// TIA Portal V16 export
// export: Created 2024-05-10T06:46:43.3869042Z, ExportSetting WithDefaults, DisplayName Totally Integrated Automation Portal, DisplayVersion V16, DisplayName TIA Portal Version Control Interface, DisplayVersion V16, DisplayName TIA Portal Openness, DisplayVersion V16, DisplayName STEP 7 Professional, DisplayVersion V16, DisplayName STEP 7 Safety, DisplayVersion V16, DisplayName WinCC Professional, DisplayVersion V16
DATA_BLOCK "K06_动作_DB"   // DB6
VERSION : 0.1
// stored: AutoNumber true, DBAccessibleFromOPCUA true, InstanceOfName K06_动作, InstanceOfType FB
"K06_动作"
   // VAR
   //    INV_Time1 : IEC_TIMER;
   //    INV_Time2 : IEC_TIMER;
   //    F100_Val_Instance1 { S7_SetPoint := 'True'} : "F100_Val";
   //    F100_Val_Instance2 { S7_SetPoint := 'True'} : "F100_Val";
   //    F100_Val_Instance3 { S7_SetPoint := 'True'} : "F100_Val";
   //    F100_Val_Instance4 { S7_SetPoint := 'True'} : "F100_Val";
   //    F100_Val_Instance5 { S7_SetPoint := 'True'} : "F100_Val";
   //    F100_Val_Instance6 { S7_SetPoint := 'True'} : "F100_Val";
   //    F100_Val_Instance7 { S7_SetPoint := 'True'} : "F100_Val";
   //    F100_Val_Instance8 { S7_SetPoint := 'True'} : "F100_Val";
   //    F100_Val_Instance9 { S7_SetPoint := 'True'} : "F100_Val";
   //    F100_Val_Instance10 { S7_SetPoint := 'True'} : "F100_Val";
   //    F100_Val_Instance11 { S7_SetPoint := 'True'} : "F100_Val";
   //    F100_Val_Instance12 { S7_SetPoint := 'True'} : "F100_Val";
   //    F100_Val_Instance13 { S7_SetPoint := 'True'} : "F100_Val";
   //    F100_Val_Instance14 { S7_SetPoint := 'True'} : "F100_Val";
   //    F100_Val_Instance15 { S7_SetPoint := 'True'} : "F100_Val";
   //    F100_Val_Instance16 { S7_SetPoint := 'True'} : "F100_Val";
   //    F100_Val_Instance17 { S7_SetPoint := 'True'} : "F100_Val";
   //    F100_Val_Instance18 { S7_SetPoint := 'True'} : "F100_Val";
   //    F100_Val_Instance19 { S7_SetPoint := 'True'} : "F100_Val";
   //    F110_Inv_Instance1 { S7_SetPoint := 'True'} : "F110_Inv";
   //    F110_Inv_Instance2 { S7_SetPoint := 'True'} : "F110_Inv";
   //    F110_Inv_Instance3 { S7_SetPoint := 'True'} : "F110_Inv";
   //    F110_Inv_Instance4 { S7_SetPoint := 'True'} : "F110_Inv";
   // END_VAR
BEGIN
END_DATA_BLOCK
